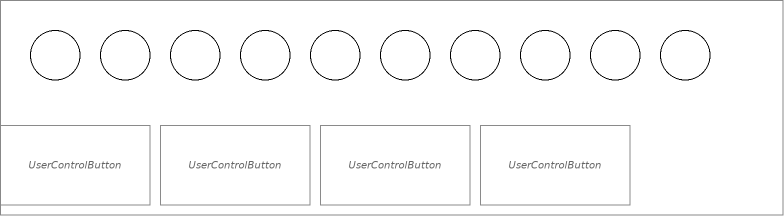
VISUALIZATION Visualization  // 784x216
    Ellipse (30,30 50x50)
        toggle MAIN.fbUnit.LED[1]
    Ellipse (100,30 50x50)
        toggle MAIN.fbUnit.LED[2]
    Ellipse (170,30 50x50)
        toggle MAIN.fbUnit.LED[3]
    Ellipse (240,30 50x50)
        toggle MAIN.fbUnit.LED[4]
    Ellipse (310,30 50x50)
        toggle MAIN.fbUnit.LED[5]
    Ellipse (380,30 50x50)
        toggle MAIN.fbUnit.LED[6]
    Ellipse (450,30 50x50)
        toggle MAIN.fbUnit.LED[7]
    Ellipse (520,30 50x50)
        toggle MAIN.fbUnit.LED[8]
    Ellipse (590,30 50x50)
        toggle MAIN.fbUnit.LED[9]
    Ellipse (660,30 50x50)
        toggle MAIN.fbUnit.LED[10]
    Polygon (783,215)
    Frame (0,125 150x80)
        shows UserControlButton(bExecute := MAIN.fbUnit.GenerateButton.bExecute, Counter := MAIN.fbUnit.GenerateButton.ExecuteCounter, sName := MAIN.fbUnit.GenerateButton.sButtonName)
    Frame (160,125 150x80)
        shows UserControlButton(bExecute := MAIN.fbUnit.ForwardButton.bExecute, Counter := MAIN.fbUnit.ForwardButton.ExecuteCounter, sName := MAIN.fbUnit.ForwardButton.sButtonName)
    Frame (320,125 150x80)
        shows UserControlButton(bExecute := MAIN.fbUnit.BackwardButton.bExecute, Counter := MAIN.fbUnit.BackwardButton.ExecuteCounter, sName := MAIN.fbUnit.BackwardButton.sButtonName)
    Frame (480,125 150x80)
        shows UserControlButton(bExecute := MAIN.fbUnit.StopButton.bExecute, Counter := MAIN.fbUnit.StopButton.ExecuteCounter, sName := MAIN.fbUnit.StopButton.sButtonName)
END_VISUALIZATION

(* stored: Version 1.1.0.1, ProductVersion 3.1.4024.12
   Visu Visualization: Id {5feb8dc8-4d54-4c59-8d10-8957f768c94c} *)
